{attribute 'TcGenerated'}
{attribute 'no-analysis'}
{attribute 'linkalways'}
// This function has been automatically generated from the project information.
VAR_GLOBAL CONSTANT
	{attribute 'const_non_replaced'}
	stLibVersion_influxdb_client : ST_LibVersion := (iMajor := 1, iMinor := 0, iBuild := 1, iRevision := 1, nFlags := 0, sVersion := '1.0.1.1');
END_VAR

(* stored: Version 1.1.0.1, ProductVersion 3.1.4024.12
   GVL Global_Version: Id {77f0868d-17ab-4334-8404-b7e47d496bdb} *)
